PROGRAM Delta_Robot_Program
VAR	
	(* Axis Enable *)
	fbEnableAxes				: FB_EnableAxes;
	io_X						: AXIS_REF;
	io_Y						: AXIS_REF;
	io_Z						: AXIS_REF;
	io_M1						: AXIS_REF;
	io_M2						: AXIS_REF;
	io_M3						: AXIS_REF;
	bEnableAxes: BOOL;
	bAllAxesReady: BOOL;
	bAxisError: BOOL;
	bResetAxes: BOOL;
	
	(* Kinematics *)
	in_stKinToPlc	AT %I*		: NCTOPLC_NCICHANNEL_REF;
	out_stPlcToKin	AT %Q*		: PLCTONC_NCICHANNEL_REF;
	fbConfigKinGroup      		: FB_KinConfigGroup;
    stAxesConfig          		: ST_KinAxes;
	fbResetKinGroup				: FB_KinResetGroup;
	bConfigKinematicGroup: BOOL;
	bUserCartesianMode: BOOL 	:= TRUE;
	bKinGroupError: BOOL;
	bResetKinematicGroup: BOOL;
	eKinematicState: E_KINSTATUS;
	bKinematicsGroupReady: BOOL;
	
	(* Jog MCS *)
	bJogEnable: BOOL;
	fbJogAxisX					: MC_Jog;
	fbJogAxisY					: MC_Jog;
	fbJogAxisZ					: MC_Jog;
	bXJogPositive: BOOL;
	bYJogPositive: BOOL;
	bZJogPositive: BOOL;
	bXJogNegative: BOOL;
	bYJogNegative: BOOL;
	bZJogNegative: BOOL;
	rJogSpeed 	 : REAL;
	
	(* Interpolation *)
	in_stItpToPlc	AT %I*		: NCTOPLC_NCICHANNEL_REF;
	out_stPlcToItp	AT %Q*		: PLCTONC_NCICHANNEL_REF;
	fUserOverRide: LREAL := 100.0;	
	fbNCIChannelGrouping: FB_NCIChannelGrouping;
	bGroupAxes: BOOL;
	bUnGroupAxes: BOOL;
	nItpState: UDINT;
	bItpError: BOOL;
	fbIntprReset : ItpResetEx2;
	bResetInteperator: BOOL;
	bNCIAxisGrouped: BOOL;
	bNCIInteperatorError: BOOL;
	fbLoadRunStop: FB_LoadFileRun;
	bRunPRogram: BOOL;
	bStopProgram: BOOL;
	sProgramName: STRING(80):='testProgram.nc';
	bNCIProgramNotRunning: BOOL;
	
	(* UI Life Bit Monitoring *)
	fbLifeBitMonitor: LifeBitMonitor;
	lifeBitStatus: BOOL;
	exception : __SYSTEM.ExceptionCode;
	bTest: bool;
END_VAR

UI();
AxisEnable();
Kinematics();
JogMCS();
NCI();

ACTION AxisEnable:
// Enable Axes
fbEnableAxes(
	bEnableAxes					:= bEnableAxes,
	bResetAxes					:= bResetAxes, 
	io_X						:= io_X , 
	io_Y						:= io_Y , 
	io_Z						:= io_Z , 
	io_M1						:= io_M1 , 
	io_M2						:= io_M2 , 
	io_M3						:= io_M3 , 
	bAllAxesReady				=> bAllAxesReady,
	bAxisError					=> bAxisError );
END_ACTION

ACTION JogMCS:
// Manual Jogging Enable after Kinematic grouping is done & NCI program is Not Running
IF bKinematicsGroupReady AND bNCIProgramNotRunning THEN
	bJogEnable := TRUE;
ELSE
	bJogEnable := FALSE;
END_IF

fbJogAxisX(
	Axis						:= io_X, 
	JogForward					:= bXJogPositive AND bJogEnable, 
	JogBackwards				:= bXJogNegative AND bJogEnable, 
	Mode						:= MC_JOGMODE_CONTINOUS,
	Velocity					:= rJogSpeed);
	
fbJogAxisY(
	Axis						:= io_Y, 
	JogForward					:= bYJogPositive AND bJogEnable, 
	JogBackwards				:= bYJogNegative AND bJogEnable, 
	Mode						:= MC_JOGMODE_CONTINOUS,
	Velocity					:= rJogSpeed);

fbJogAxisZ(
	Axis						:= io_Z, 
	JogForward					:= bZJogPositive AND bJogEnable, 
	JogBackwards				:= bZJogNegative AND bJogEnable, 
	Mode						:= MC_JOGMODE_CONTINOUS,
	Velocity					:= rJogSpeed);
END_ACTION

ACTION Kinematics:
// Read axes id's from cylic interface
// so they can be mapped later to the kinematic group
stAxesConfig.nAxisIdsAcs[1]		:= io_M1.NcToPlc.AxisId;
stAxesConfig.nAxisIdsAcs[2]		:= io_M2.NcToPlc.AxisId;
stAxesConfig.nAxisIdsAcs[3]		:= io_M3.NcToPlc.AxisId;
stAxesConfig.nAxisIdsMcs[1]		:= io_X.NcToPlc.AxisId;
stAxesConfig.nAxisIdsMcs[2]		:= io_Y.NcToPlc.AxisId;
stAxesConfig.nAxisIdsMcs[3]		:= io_Z.NcToPlc.AxisId;

//Read Kinematics Status
eKinematicState := F_KinGetChnOperationState(stKinRefIn:=in_stKinToPlc);
IF eKinematicState = E_KINSTATUS.KinStatus_Ready THEN
	bKinematicsGroupReady := TRUE;
	bKinGroupError := FALSE;
ELSIF eKinematicState = E_KINSTATUS.KinStatus_Error THEN 
	bKinGroupError := TRUE;
	bKinematicsGroupReady := FALSE;
ELSE
	bKinematicsGroupReady := FALSE;
	bKinGroupError := FALSE	;
END_IF


// Build Kinematic Group
fbConfigKinGroup(
	bExecute					:= bConfigKinematicGroup AND bAllAxesReady AND NOT bAxisError , 
	bCartesianMode				:= bUserCartesianMode, 
	stAxesList					:= stAxesConfig, 
	stKinRefIn					:= in_stKinToPlc);

//Reset Kinematic Group
fbResetKinGroup(
	bExecute					:= bResetKinematicGroup , 
	nItpChannelId				:= in_stKinToPlc.ChnId, 
	stKinRefIn					:= in_stKinToPlc, 
	stAxesList					:= stAxesConfig);
END_ACTION

ACTION NCI:
(* Set OverRide % *)
ItpSetOverridePercent(fOverridePercent := fUserOverRide,sPlcToNci:=out_stPlcToItp);

(* Grouping Axis *)
fbNCIChannelGrouping(
	bGroupChannel:= bGroupAxes AND bKinematicsGroupReady AND bAllAxesReady AND NOT bAxisError AND NOT bItpError, 
	bUnGroupChannel:= bUnGroupAxes, 
	stX:=io_X, 
	stY:=io_Y, 
	stZ:=io_Z, 
	stItpToPlc:=in_stItpToPlc, 
	stPlcToItp:=out_stPlcToItp, 
	bBusy=> , 
	bError=> , 
	bDone=>bNCIAxisGrouped);
	
(* Inteperator State *)
nItpState := ItpGetStateInterpreter( in_stItpToPlc ); 

(* Inteperator Error *)
bNCIInteperatorError := bItpError := ItpHasError( in_stItpToPlc ); 

(* Reset Inteperator *)
fbIntprReset(
	bExecute:=bResetInteperator, 
	tTimeOut:= , 
	sNciToPlc:=in_stItpToPlc, 
	bBusy=> , 
	bErr=> , 
	nErrId=> );
	
(* Program Run & Stop NCI Program from File *)
fbLoadRunStop(
	bRun:=bRunPRogram,
	bStop :=bStopProgram,
	sPrgName:=sProgramName, 
	stItpToPlc:=in_stItpToPlc, 
	stPlcToItp:=out_stPlcToItp, 
	bBusy=> , 
	bDone=> , 
	bError=> , 
	nInterpreterState=> );
	
(* Interlock for Jog *)
IF nItpState = 1 OR nItpState = 2 THEN
	bNCIProgramNotRunning := TRUE;
ELSE
	bNCIProgramNotRunning := FALSE;
END_IF
END_ACTION

ACTION UI:
(* Life Bit Monitoring *)
IF UIData.stUI_TO_PLC.EnableMonitoring THEN
	fbLifeBitMonitor.MonitoringTime := T#800MS;
	fbLifeBitMonitor.StartMonitor();
ELSE
	fbLifeBitMonitor.StopMonitor();
END_IF

lifeBitStatus := fbLifeBitMonitor.Status(LifeBit:=UIData.stUI_TO_PLC.LifeBit);

IF NOT lifeBitStatus THEN
	(* For __TRY __CATCH Supported Platform *)
	(*
	__TRY
		MEMSET(destAddr:=ADR(UIData.stUI_TO_PLC.LifeBit),
		   	   fillByte:=16#0,
		   	   n:=SIZEOF(UIData.stUI_TO_PLC)-1); //SIZE - 1 is Enable Monitoring Bit size deleted
	__CATCH(exception)
			//In case of Error 
	__ENDTRY 
	*)	
	UIData.stUI_TO_PLC.EnableMonitoring:=UIData.stUI_TO_PLC.LifeBit := 0;
	UIData.stUI_TO_PLC.EnableAllAxis:= UIData.stUI_TO_PLC.ResetAllAxis:= 0;
	UIData.stUI_TO_PLC.ConfigKinematicGroup:= UIData.stUI_TO_PLC.ResetKinematicGroup := 0;
	UIData.stUI_TO_PLC.XJogPositive := UIData.stUI_TO_PLC.YJogPositive := 0;
	UIData.stUI_TO_PLC.ZJogPositive := UIData.stUI_TO_PLC.XJogNegative := 0;
	UIData.stUI_TO_PLC.YJogNegative := UIData.stUI_TO_PLC.ZJogNegative:= 0;
	UIData.stUI_TO_PLC.JogSpeed := 0;
	UIData.stUI_TO_PLC.NCIAxisGroup:= 0;
	UIData.stUI_TO_PLC.NCIAxisUnGroup := UIData.stUI_TO_PLC.NCIInteperatorReset:= 0;
	UIData.stUI_TO_PLC.RunPartProgram := UIData.stUI_TO_PLC.StopPartProgram:= 0;
	UIData.stUI_TO_PLC.NCIOverRidePer := 0;
	UIData.stUI_TO_PLC.PartProgramName:= '';
	
END_IF

(*PLC to UI*)

//Position Data
UIData.stPLC_TO_UI.X_MCSPos := io_X.NcToPlc.ActPos;
UIData.stPLC_TO_UI.Y_MCSPos := io_Y.NcToPlc.ActPos;
UIData.stPLC_TO_UI.Z_MCSPos := io_Z.NcToPlc.ActPos;
UIData.stPLC_TO_UI.M1_ACSPos := io_M1.NcToPlc.ActPos;
UIData.stPLC_TO_UI.M2_ACSPos := io_M2.NcToPlc.ActPos;
UIData.stPLC_TO_UI.M3_ACSPos := io_M3.NcToPlc.ActPos;

//Axis Status
UIData.stPLC_TO_UI.AllAxisEnabled := bAllAxesReady; 
UIData.stPLC_TO_UI.AxisError := bAxisError; 
UIData.stPLC_TO_UI.KinematicGroupError := bKinGroupError;

//Kinematic Status
UIData.stPLC_TO_UI.KinematicGroupingReady := bKinematicsGroupReady;
UIData.stPLC_TO_UI.KinematicGroupError := bKinGroupError;
UIData.stPLC_TO_UI.NCIAxisGrouped := bNCIAxisGrouped;
UIData.stPLC_TO_UI.NCIAXisError := bNCIInteperatorError;
UIData.stPLC_TO_UI.NCIInterpreterState := nItpState;

(*UI to PLC*)
bEnableAxes := UIData.stUI_TO_PLC.EnableAllAxis;
bResetAxes := UIData.stUI_TO_PLC.ResetAllAxis;
bConfigKinematicGroup := UIData.stUI_TO_PLC.ConfigKinematicGroup;
bResetKinematicGroup := UIData.stUI_TO_PLC.ResetKinematicGroup;
bXJogPositive := UIData.stUI_TO_PLC.XJogPositive;
bYJogPositive := UIData.stUI_TO_PLC.YJogPositive;
bZJogPositive := UIData.stUI_TO_PLC.ZJogPositive;
bXJogNegative := UIData.stUI_TO_PLC.XJogNegative;
bYJogNegative := UIData.stUI_TO_PLC.YJogNegative;
bZJogNegative := UIData.stUI_TO_PLC.ZJogNegative;
rJogSpeed     := UIData.stUI_TO_PLC.JogSpeed;
bGroupAxes 	  := UIData.stUI_TO_PLC.NCIAxisGroup;
bUnGroupAxes  := UIData.stUI_TO_PLC.NCIAxisUnGroup;
bResetInteperator := UIData.stUI_TO_PLC.NCIInteperatorReset;
bRunPRogram 	  := UIData.stUI_TO_PLC.RunPartProgram;
bStopProgram 	  := UIData.stUI_TO_PLC.StopPartProgram;
fUserOverRide 	:= UIData.stUI_TO_PLC.NCIOverRidePer;
sProgramName := UIData.stUI_TO_PLC.PartProgramName;
END_ACTION

END_PROGRAM

(* stored: Version 1.1.0.1, ProductVersion 3.1.4024.12
   POU Delta_Robot_Program: Id {ec9c67e2-5b7f-42f3-9848-db5938141bd5}, SpecialFunc None
   Action AxisEnable: Id {19d5fb57-971b-4542-8d41-9f4bffbdae44}
   Action JogMCS: Id {773da444-5073-46a7-a95b-c0c675e8c1cf}
   Action Kinematics: Id {df827e87-35b7-4c3a-95a4-782f5599478c}
   Action NCI: Id {6a955fd0-4f1a-4d83-9d56-fe86d51094c4}
   Action UI: Id {62a58446-a97c-4afd-920b-3f96fac39f08} *)
